DATA_BLOCK "DB2010_V"
TITLE = DB2010_V
{ S7_Optimized_Access := 'FALSE' }
AUTHOR : ABH
FAMILY : ZeusControl
VERSION : 1.0
//Bloique de datos valvula.
   STRUCT
      V { S7_SetPoint := 'False'} : Array[0.."N_MAX_DISP_V"] of "ZC_DISP_V";
      Mux { S7_SetPoint := 'False'} : Array[0.."N_MAX_MUX_DISP"] of "ZC_DISP_MUX_V";
      Agrup : Array[0.."N_MAX_DISP_AGRUP"] of "ZC_DISP_AGRUP";
   END_STRUCT;


BEGIN
   V[0].Hmi_Nombre := '';
   V[0].Hmi_Estado := 0;
   V[0].Estado_AutoMan := FALSE;
   V[0].Estado_Activado := FALSE;
   V[0].Estado_Enclavado := FALSE;
   V[0].Estado_EntradaRetornoReposo := FALSE;
   V[0].Estado_EntradaRetornoTrabajo := FALSE;
   V[0].Alarmas_Reposo := FALSE;
   V[0].Alarmas_Trabajo := FALSE;
   V[0].Alarmas_Mantenimiento := FALSE;
   V[0].Alarmas_Doble := FALSE;
   V[0].Alarmas_General := FALSE;
   V[0].Orden_ActivarManual := FALSE;
   V[0].Orden_ActivarAuto := TRUE;
   V[0].Orden_ResetCiclos := FALSE;
   V[0].Config_Habilitar := FALSE;
   V[0].Config_HabilitarRetornoReposo := TRUE;
   V[0].Config_HabilitarInvertirReposo := FALSE;
   V[0].Config_HabilitarRetornoTrabajo := TRUE;
   V[0].Config_HabilitarInvertirTrabajo := FALSE;
   V[0].Config_HabilitarMantenimiento := FALSE;
   V[0].Aux_oldActivado := FALSE;
   V[0].Aux_oldAlarma := FALSE;
   V[0].Aux_oldAutoMan := FALSE;
   V[0].Estado_SeguridadOk := TRUE;
   V[0].Config_GrupoAlarma := 0;
   V[0].Config_DireccionSalidaByte := 0;
   V[0].Config_DireccionSalidaBit := 0;
   V[0].Config_DireccionRetReposoByte := 0;
   V[0].Config_DireccionRetReposoBit := 0;
   V[0].Config_DireccionRetTrabajoByte := 0;
   V[0].Config_DireccionRetTrabajoBit := 0;
   V[0].Tiempos_SetPointTiempoAlarma := 10;
   V[0].Tiempos_Alarma := 0;
   V[0].Tiempos_SetPointCiclos := 1000;
   V[0].Tiempos_Ciclos := 0;
   V[1].Hmi_Nombre := 'VA-101';
   V[1].Hmi_Estado := 1;
   V[1].Estado_AutoMan := FALSE;
   V[1].Estado_Activado := FALSE;
   V[1].Estado_Enclavado := FALSE;
   V[1].Estado_EntradaRetornoReposo := FALSE;
   V[1].Estado_EntradaRetornoTrabajo := FALSE;
   V[1].Alarmas_Reposo := FALSE;
   V[1].Alarmas_Trabajo := FALSE;
   V[1].Alarmas_Mantenimiento := FALSE;
   V[1].Alarmas_Doble := FALSE;
   V[1].Alarmas_General := FALSE;
   V[1].Orden_ActivarManual := FALSE;
   V[1].Orden_ActivarAuto := FALSE;
   V[1].Orden_ResetCiclos := FALSE;
   V[1].Config_Habilitar := TRUE;
   V[1].Config_HabilitarRetornoReposo := FALSE;
   V[1].Config_HabilitarInvertirReposo := FALSE;
   V[1].Config_HabilitarRetornoTrabajo := TRUE;
   V[1].Config_HabilitarInvertirTrabajo := FALSE;
   V[1].Config_HabilitarMantenimiento := FALSE;
   V[1].Aux_oldActivado := FALSE;
   V[1].Aux_oldAlarma := FALSE;
   V[1].Aux_oldAutoMan := FALSE;
   V[1].Estado_SeguridadOk := TRUE;
   V[1].Config_GrupoAlarma := 0;
   V[1].Config_DireccionSalidaByte := 102;
   V[1].Config_DireccionSalidaBit := 0;
   V[1].Config_DireccionRetReposoByte := 0;
   V[1].Config_DireccionRetReposoBit := 0;
   V[1].Config_DireccionRetTrabajoByte := 102;
   V[1].Config_DireccionRetTrabajoBit := 0;
   V[1].Tiempos_SetPointTiempoAlarma := 10;
   V[1].Tiempos_Alarma := 0;
   V[1].Tiempos_SetPointCiclos := 1000;
   V[1].Tiempos_Ciclos := 66;
   V[2].Hmi_Nombre := 'VA-102';
   V[2].Hmi_Estado := 1;
   V[2].Estado_AutoMan := FALSE;
   V[2].Estado_Activado := FALSE;
   V[2].Estado_Enclavado := FALSE;
   V[2].Estado_EntradaRetornoReposo := FALSE;
   V[2].Estado_EntradaRetornoTrabajo := FALSE;
   V[2].Alarmas_Reposo := FALSE;
   V[2].Alarmas_Trabajo := FALSE;
   V[2].Alarmas_Mantenimiento := FALSE;
   V[2].Alarmas_Doble := FALSE;
   V[2].Alarmas_General := FALSE;
   V[2].Orden_ActivarManual := FALSE;
   V[2].Orden_ActivarAuto := FALSE;
   V[2].Orden_ResetCiclos := FALSE;
   V[2].Config_Habilitar := TRUE;
   V[2].Config_HabilitarRetornoReposo := FALSE;
   V[2].Config_HabilitarInvertirReposo := FALSE;
   V[2].Config_HabilitarRetornoTrabajo := TRUE;
   V[2].Config_HabilitarInvertirTrabajo := FALSE;
   V[2].Config_HabilitarMantenimiento := FALSE;
   V[2].Aux_oldActivado := FALSE;
   V[2].Aux_oldAlarma := FALSE;
   V[2].Aux_oldAutoMan := FALSE;
   V[2].Estado_SeguridadOk := TRUE;
   V[2].Config_GrupoAlarma := 0;
   V[2].Config_DireccionSalidaByte := 102;
   V[2].Config_DireccionSalidaBit := 1;
   V[2].Config_DireccionRetReposoByte := 0;
   V[2].Config_DireccionRetReposoBit := 0;
   V[2].Config_DireccionRetTrabajoByte := 102;
   V[2].Config_DireccionRetTrabajoBit := 1;
   V[2].Tiempos_SetPointTiempoAlarma := 10;
   V[2].Tiempos_Alarma := 0;
   V[2].Tiempos_SetPointCiclos := 1000;
   V[2].Tiempos_Ciclos := 104;
   V[3].Hmi_Nombre := 'VAD-103';
   V[3].Hmi_Estado := 1;
   V[3].Estado_AutoMan := FALSE;
   V[3].Estado_Activado := FALSE;
   V[3].Estado_Enclavado := FALSE;
   V[3].Estado_EntradaRetornoReposo := FALSE;
   V[3].Estado_EntradaRetornoTrabajo := FALSE;
   V[3].Alarmas_Reposo := FALSE;
   V[3].Alarmas_Trabajo := FALSE;
   V[3].Alarmas_Mantenimiento := FALSE;
   V[3].Alarmas_Doble := FALSE;
   V[3].Alarmas_General := FALSE;
   V[3].Orden_ActivarManual := FALSE;
   V[3].Orden_ActivarAuto := FALSE;
   V[3].Orden_ResetCiclos := FALSE;
   V[3].Config_Habilitar := TRUE;
   V[3].Config_HabilitarRetornoReposo := FALSE;
   V[3].Config_HabilitarInvertirReposo := FALSE;
   V[3].Config_HabilitarRetornoTrabajo := TRUE;
   V[3].Config_HabilitarInvertirTrabajo := FALSE;
   V[3].Config_HabilitarMantenimiento := FALSE;
   V[3].Aux_oldActivado := FALSE;
   V[3].Aux_oldAlarma := FALSE;
   V[3].Aux_oldAutoMan := FALSE;
   V[3].Estado_SeguridadOk := TRUE;
   V[3].Config_GrupoAlarma := 0;
   V[3].Config_DireccionSalidaByte := 102;
   V[3].Config_DireccionSalidaBit := 2;
   V[3].Config_DireccionRetReposoByte := 0;
   V[3].Config_DireccionRetReposoBit := 0;
   V[3].Config_DireccionRetTrabajoByte := 102;
   V[3].Config_DireccionRetTrabajoBit := 2;
   V[3].Tiempos_SetPointTiempoAlarma := 10;
   V[3].Tiempos_Alarma := 0;
   V[3].Tiempos_SetPointCiclos := 1000;
   V[3].Tiempos_Ciclos := 118;
   V[4].Hmi_Nombre := 'VAD-108';
   V[4].Hmi_Estado := 1;
   V[4].Estado_AutoMan := FALSE;
   V[4].Estado_Activado := FALSE;
   V[4].Estado_Enclavado := FALSE;
   V[4].Estado_EntradaRetornoReposo := FALSE;
   V[4].Estado_EntradaRetornoTrabajo := FALSE;
   V[4].Alarmas_Reposo := FALSE;
   V[4].Alarmas_Trabajo := FALSE;
   V[4].Alarmas_Mantenimiento := FALSE;
   V[4].Alarmas_Doble := FALSE;
   V[4].Alarmas_General := FALSE;
   V[4].Orden_ActivarManual := FALSE;
   V[4].Orden_ActivarAuto := FALSE;
   V[4].Orden_ResetCiclos := FALSE;
   V[4].Config_Habilitar := TRUE;
   V[4].Config_HabilitarRetornoReposo := FALSE;
   V[4].Config_HabilitarInvertirReposo := FALSE;
   V[4].Config_HabilitarRetornoTrabajo := TRUE;
   V[4].Config_HabilitarInvertirTrabajo := FALSE;
   V[4].Config_HabilitarMantenimiento := FALSE;
   V[4].Aux_oldActivado := FALSE;
   V[4].Aux_oldAlarma := FALSE;
   V[4].Aux_oldAutoMan := FALSE;
   V[4].Estado_SeguridadOk := TRUE;
   V[4].Config_GrupoAlarma := 0;
   V[4].Config_DireccionSalidaByte := 102;
   V[4].Config_DireccionSalidaBit := 3;
   V[4].Config_DireccionRetReposoByte := 0;
   V[4].Config_DireccionRetReposoBit := 0;
   V[4].Config_DireccionRetTrabajoByte := 102;
   V[4].Config_DireccionRetTrabajoBit := 3;
   V[4].Tiempos_SetPointTiempoAlarma := 10;
   V[4].Tiempos_Alarma := 0;
   V[4].Tiempos_SetPointCiclos := 1000;
   V[4].Tiempos_Ciclos := 28;
   V[5].Hmi_Nombre := 'VA-114';
   V[5].Hmi_Estado := 1;
   V[5].Estado_AutoMan := FALSE;
   V[5].Estado_Activado := FALSE;
   V[5].Estado_Enclavado := FALSE;
   V[5].Estado_EntradaRetornoReposo := FALSE;
   V[5].Estado_EntradaRetornoTrabajo := FALSE;
   V[5].Alarmas_Reposo := FALSE;
   V[5].Alarmas_Trabajo := FALSE;
   V[5].Alarmas_Mantenimiento := FALSE;
   V[5].Alarmas_Doble := FALSE;
   V[5].Alarmas_General := FALSE;
   V[5].Orden_ActivarManual := FALSE;
   V[5].Orden_ActivarAuto := FALSE;
   V[5].Orden_ResetCiclos := FALSE;
   V[5].Config_Habilitar := TRUE;
   V[5].Config_HabilitarRetornoReposo := FALSE;
   V[5].Config_HabilitarInvertirReposo := FALSE;
   V[5].Config_HabilitarRetornoTrabajo := TRUE;
   V[5].Config_HabilitarInvertirTrabajo := FALSE;
   V[5].Config_HabilitarMantenimiento := FALSE;
   V[5].Aux_oldActivado := FALSE;
   V[5].Aux_oldAlarma := FALSE;
   V[5].Aux_oldAutoMan := FALSE;
   V[5].Estado_SeguridadOk := TRUE;
   V[5].Config_GrupoAlarma := 0;
   V[5].Config_DireccionSalidaByte := 102;
   V[5].Config_DireccionSalidaBit := 4;
   V[5].Config_DireccionRetReposoByte := 0;
   V[5].Config_DireccionRetReposoBit := 0;
   V[5].Config_DireccionRetTrabajoByte := 102;
   V[5].Config_DireccionRetTrabajoBit := 4;
   V[5].Tiempos_SetPointTiempoAlarma := 10;
   V[5].Tiempos_Alarma := 0;
   V[5].Tiempos_SetPointCiclos := 1000;
   V[5].Tiempos_Ciclos := 6;
   V[6].Hmi_Nombre := 'VA3-115';
   V[6].Hmi_Estado := 1;
   V[6].Estado_AutoMan := FALSE;
   V[6].Estado_Activado := FALSE;
   V[6].Estado_Enclavado := FALSE;
   V[6].Estado_EntradaRetornoReposo := FALSE;
   V[6].Estado_EntradaRetornoTrabajo := FALSE;
   V[6].Alarmas_Reposo := FALSE;
   V[6].Alarmas_Trabajo := FALSE;
   V[6].Alarmas_Mantenimiento := FALSE;
   V[6].Alarmas_Doble := FALSE;
   V[6].Alarmas_General := FALSE;
   V[6].Orden_ActivarManual := FALSE;
   V[6].Orden_ActivarAuto := FALSE;
   V[6].Orden_ResetCiclos := FALSE;
   V[6].Config_Habilitar := TRUE;
   V[6].Config_HabilitarRetornoReposo := FALSE;
   V[6].Config_HabilitarInvertirReposo := FALSE;
   V[6].Config_HabilitarRetornoTrabajo := TRUE;
   V[6].Config_HabilitarInvertirTrabajo := FALSE;
   V[6].Config_HabilitarMantenimiento := FALSE;
   V[6].Aux_oldActivado := FALSE;
   V[6].Aux_oldAlarma := FALSE;
   V[6].Aux_oldAutoMan := FALSE;
   V[6].Estado_SeguridadOk := TRUE;
   V[6].Config_GrupoAlarma := 0;
   V[6].Config_DireccionSalidaByte := 102;
   V[6].Config_DireccionSalidaBit := 5;
   V[6].Config_DireccionRetReposoByte := 0;
   V[6].Config_DireccionRetReposoBit := 0;
   V[6].Config_DireccionRetTrabajoByte := 102;
   V[6].Config_DireccionRetTrabajoBit := 5;
   V[6].Tiempos_SetPointTiempoAlarma := 10;
   V[6].Tiempos_Alarma := 0;
   V[6].Tiempos_SetPointCiclos := 1000;
   V[6].Tiempos_Ciclos := 6;
   V[7].Hmi_Nombre := 'VA3-116';
   V[7].Hmi_Estado := 1;
   V[7].Estado_AutoMan := FALSE;
   V[7].Estado_Activado := FALSE;
   V[7].Estado_Enclavado := FALSE;
   V[7].Estado_EntradaRetornoReposo := FALSE;
   V[7].Estado_EntradaRetornoTrabajo := FALSE;
   V[7].Alarmas_Reposo := FALSE;
   V[7].Alarmas_Trabajo := FALSE;
   V[7].Alarmas_Mantenimiento := FALSE;
   V[7].Alarmas_Doble := FALSE;
   V[7].Alarmas_General := FALSE;
   V[7].Orden_ActivarManual := FALSE;
   V[7].Orden_ActivarAuto := FALSE;
   V[7].Orden_ResetCiclos := FALSE;
   V[7].Config_Habilitar := TRUE;
   V[7].Config_HabilitarRetornoReposo := FALSE;
   V[7].Config_HabilitarInvertirReposo := FALSE;
   V[7].Config_HabilitarRetornoTrabajo := TRUE;
   V[7].Config_HabilitarInvertirTrabajo := FALSE;
   V[7].Config_HabilitarMantenimiento := FALSE;
   V[7].Aux_oldActivado := FALSE;
   V[7].Aux_oldAlarma := FALSE;
   V[7].Aux_oldAutoMan := FALSE;
   V[7].Estado_SeguridadOk := TRUE;
   V[7].Config_GrupoAlarma := 0;
   V[7].Config_DireccionSalidaByte := 102;
   V[7].Config_DireccionSalidaBit := 6;
   V[7].Config_DireccionRetReposoByte := 0;
   V[7].Config_DireccionRetReposoBit := 0;
   V[7].Config_DireccionRetTrabajoByte := 102;
   V[7].Config_DireccionRetTrabajoBit := 6;
   V[7].Tiempos_SetPointTiempoAlarma := 10;
   V[7].Tiempos_Alarma := 0;
   V[7].Tiempos_SetPointCiclos := 1000;
   V[7].Tiempos_Ciclos := 6;
   V[8].Hmi_Nombre := 'VAD-117';
   V[8].Hmi_Estado := 1;
   V[8].Estado_AutoMan := FALSE;
   V[8].Estado_Activado := FALSE;
   V[8].Estado_Enclavado := FALSE;
   V[8].Estado_EntradaRetornoReposo := FALSE;
   V[8].Estado_EntradaRetornoTrabajo := FALSE;
   V[8].Alarmas_Reposo := FALSE;
   V[8].Alarmas_Trabajo := FALSE;
   V[8].Alarmas_Mantenimiento := FALSE;
   V[8].Alarmas_Doble := FALSE;
   V[8].Alarmas_General := FALSE;
   V[8].Orden_ActivarManual := FALSE;
   V[8].Orden_ActivarAuto := FALSE;
   V[8].Orden_ResetCiclos := FALSE;
   V[8].Config_Habilitar := TRUE;
   V[8].Config_HabilitarRetornoReposo := FALSE;
   V[8].Config_HabilitarInvertirReposo := FALSE;
   V[8].Config_HabilitarRetornoTrabajo := TRUE;
   V[8].Config_HabilitarInvertirTrabajo := FALSE;
   V[8].Config_HabilitarMantenimiento := FALSE;
   V[8].Aux_oldActivado := FALSE;
   V[8].Aux_oldAlarma := FALSE;
   V[8].Aux_oldAutoMan := FALSE;
   V[8].Estado_SeguridadOk := TRUE;
   V[8].Config_GrupoAlarma := 0;
   V[8].Config_DireccionSalidaByte := 102;
   V[8].Config_DireccionSalidaBit := 7;
   V[8].Config_DireccionRetReposoByte := 0;
   V[8].Config_DireccionRetReposoBit := 0;
   V[8].Config_DireccionRetTrabajoByte := 102;
   V[8].Config_DireccionRetTrabajoBit := 7;
   V[8].Tiempos_SetPointTiempoAlarma := 10;
   V[8].Tiempos_Alarma := 0;
   V[8].Tiempos_SetPointCiclos := 1000;
   V[8].Tiempos_Ciclos := 84;
   V[9].Hmi_Nombre := 'VAD-120';
   V[9].Hmi_Estado := 1;
   V[9].Estado_AutoMan := FALSE;
   V[9].Estado_Activado := FALSE;
   V[9].Estado_Enclavado := FALSE;
   V[9].Estado_EntradaRetornoReposo := FALSE;
   V[9].Estado_EntradaRetornoTrabajo := FALSE;
   V[9].Alarmas_Reposo := FALSE;
   V[9].Alarmas_Trabajo := FALSE;
   V[9].Alarmas_Mantenimiento := FALSE;
   V[9].Alarmas_Doble := FALSE;
   V[9].Alarmas_General := FALSE;
   V[9].Orden_ActivarManual := FALSE;
   V[9].Orden_ActivarAuto := FALSE;
   V[9].Orden_ResetCiclos := FALSE;
   V[9].Config_Habilitar := TRUE;
   V[9].Config_HabilitarRetornoReposo := FALSE;
   V[9].Config_HabilitarInvertirReposo := FALSE;
   V[9].Config_HabilitarRetornoTrabajo := TRUE;
   V[9].Config_HabilitarInvertirTrabajo := FALSE;
   V[9].Config_HabilitarMantenimiento := FALSE;
   V[9].Aux_oldActivado := FALSE;
   V[9].Aux_oldAlarma := FALSE;
   V[9].Aux_oldAutoMan := FALSE;
   V[9].Estado_SeguridadOk := TRUE;
   V[9].Config_GrupoAlarma := 0;
   V[9].Config_DireccionSalidaByte := 103;
   V[9].Config_DireccionSalidaBit := 0;
   V[9].Config_DireccionRetReposoByte := 0;
   V[9].Config_DireccionRetReposoBit := 0;
   V[9].Config_DireccionRetTrabajoByte := 103;
   V[9].Config_DireccionRetTrabajoBit := 0;
   V[9].Tiempos_SetPointTiempoAlarma := 10;
   V[9].Tiempos_Alarma := 0;
   V[9].Tiempos_SetPointCiclos := 1000;
   V[9].Tiempos_Ciclos := 28;
   V[10].Hmi_Nombre := 'VA-126';
   V[10].Hmi_Estado := 1;
   V[10].Estado_AutoMan := FALSE;
   V[10].Estado_Activado := FALSE;
   V[10].Estado_Enclavado := FALSE;
   V[10].Estado_EntradaRetornoReposo := FALSE;
   V[10].Estado_EntradaRetornoTrabajo := FALSE;
   V[10].Alarmas_Reposo := FALSE;
   V[10].Alarmas_Trabajo := FALSE;
   V[10].Alarmas_Mantenimiento := FALSE;
   V[10].Alarmas_Doble := FALSE;
   V[10].Alarmas_General := FALSE;
   V[10].Orden_ActivarManual := FALSE;
   V[10].Orden_ActivarAuto := FALSE;
   V[10].Orden_ResetCiclos := FALSE;
   V[10].Config_Habilitar := TRUE;
   V[10].Config_HabilitarRetornoReposo := FALSE;
   V[10].Config_HabilitarInvertirReposo := FALSE;
   V[10].Config_HabilitarRetornoTrabajo := TRUE;
   V[10].Config_HabilitarInvertirTrabajo := FALSE;
   V[10].Config_HabilitarMantenimiento := FALSE;
   V[10].Aux_oldActivado := FALSE;
   V[10].Aux_oldAlarma := FALSE;
   V[10].Aux_oldAutoMan := FALSE;
   V[10].Estado_SeguridadOk := TRUE;
   V[10].Config_GrupoAlarma := 0;
   V[10].Config_DireccionSalidaByte := 103;
   V[10].Config_DireccionSalidaBit := 1;
   V[10].Config_DireccionRetReposoByte := 0;
   V[10].Config_DireccionRetReposoBit := 0;
   V[10].Config_DireccionRetTrabajoByte := 103;
   V[10].Config_DireccionRetTrabajoBit := 1;
   V[10].Tiempos_SetPointTiempoAlarma := 10;
   V[10].Tiempos_Alarma := 0;
   V[10].Tiempos_SetPointCiclos := 1000;
   V[10].Tiempos_Ciclos := 70;
   Mux[0].Habilitar := TRUE;
   Mux[0].ExisteCambio := FALSE;
   Mux[0].MaxVisible := FALSE;
   Mux[0].Index := 182;
   Mux[0].oldIndex := 182;
   Mux[0].V.Hmi_Nombre := 'VA-438';
   Mux[0].V.Hmi_Estado := 1;
   Mux[0].V.Estado_AutoMan := FALSE;
   Mux[0].V.Estado_Activado := FALSE;
   Mux[0].V.Estado_Enclavado := FALSE;
   Mux[0].V.Estado_EntradaRetornoReposo := FALSE;
   Mux[0].V.Estado_EntradaRetornoTrabajo := FALSE;
   Mux[0].V.Alarmas_Reposo := FALSE;
   Mux[0].V.Alarmas_Trabajo := FALSE;
   Mux[0].V.Alarmas_Mantenimiento := FALSE;
   Mux[0].V.Alarmas_Doble := FALSE;
   Mux[0].V.Alarmas_General := FALSE;
   Mux[0].V.Orden_ActivarManual := FALSE;
   Mux[0].V.Orden_ActivarAuto := FALSE;
   Mux[0].V.Orden_ResetCiclos := FALSE;
   Mux[0].V.Config_Habilitar := TRUE;
   Mux[0].V.Config_HabilitarRetornoReposo := FALSE;
   Mux[0].V.Config_HabilitarInvertirReposo := FALSE;
   Mux[0].V.Config_HabilitarRetornoTrabajo := FALSE;
   Mux[0].V.Config_HabilitarInvertirTrabajo := FALSE;
   Mux[0].V.Config_HabilitarMantenimiento := FALSE;
   Mux[0].V.Aux_oldActivado := FALSE;
   Mux[0].V.Aux_oldAlarma := FALSE;
   Mux[0].V.Aux_oldAutoMan := FALSE;
   Mux[0].V.Estado_SeguridadOk := TRUE;
   Mux[0].V.Config_GrupoAlarma := 2;
   Mux[0].V.Config_DireccionSalidaByte := 325;
   Mux[0].V.Config_DireccionSalidaBit := 2;
   Mux[0].V.Config_DireccionRetReposoByte := 0;
   Mux[0].V.Config_DireccionRetReposoBit := 0;
   Mux[0].V.Config_DireccionRetTrabajoByte := 0;
   Mux[0].V.Config_DireccionRetTrabajoBit := 0;
   Mux[0].V.Tiempos_SetPointTiempoAlarma := 10;
   Mux[0].V.Tiempos_Alarma := 0;
   Mux[0].V.Tiempos_SetPointCiclos := 1000;
   Mux[0].V.Tiempos_Ciclos := 1200;
   Mux[1].Habilitar := TRUE;
   Mux[1].ExisteCambio := FALSE;
   Mux[1].MaxVisible := FALSE;
   Mux[1].Index := 0;
   Mux[1].oldIndex := 0;
   Mux[1].V.Hmi_Nombre := '';
   Mux[1].V.Hmi_Estado := 0;
   Mux[1].V.Estado_AutoMan := FALSE;
   Mux[1].V.Estado_Activado := FALSE;
   Mux[1].V.Estado_Enclavado := FALSE;
   Mux[1].V.Estado_EntradaRetornoReposo := FALSE;
   Mux[1].V.Estado_EntradaRetornoTrabajo := FALSE;
   Mux[1].V.Alarmas_Reposo := FALSE;
   Mux[1].V.Alarmas_Trabajo := FALSE;
   Mux[1].V.Alarmas_Mantenimiento := FALSE;
   Mux[1].V.Alarmas_Doble := FALSE;
   Mux[1].V.Alarmas_General := FALSE;
   Mux[1].V.Orden_ActivarManual := FALSE;
   Mux[1].V.Orden_ActivarAuto := TRUE;
   Mux[1].V.Orden_ResetCiclos := FALSE;
   Mux[1].V.Config_Habilitar := FALSE;
   Mux[1].V.Config_HabilitarRetornoReposo := TRUE;
   Mux[1].V.Config_HabilitarInvertirReposo := FALSE;
   Mux[1].V.Config_HabilitarRetornoTrabajo := TRUE;
   Mux[1].V.Config_HabilitarInvertirTrabajo := FALSE;
   Mux[1].V.Config_HabilitarMantenimiento := FALSE;
   Mux[1].V.Aux_oldActivado := FALSE;
   Mux[1].V.Aux_oldAlarma := FALSE;
   Mux[1].V.Aux_oldAutoMan := FALSE;
   Mux[1].V.Estado_SeguridadOk := TRUE;
   Mux[1].V.Config_GrupoAlarma := 0;
   Mux[1].V.Config_DireccionSalidaByte := 0;
   Mux[1].V.Config_DireccionSalidaBit := 0;
   Mux[1].V.Config_DireccionRetReposoByte := 0;
   Mux[1].V.Config_DireccionRetReposoBit := 0;
   Mux[1].V.Config_DireccionRetTrabajoByte := 0;
   Mux[1].V.Config_DireccionRetTrabajoBit := 0;
   Mux[1].V.Tiempos_SetPointTiempoAlarma := 10;
   Mux[1].V.Tiempos_Alarma := 0;
   Mux[1].V.Tiempos_SetPointCiclos := 1000;
   Mux[1].V.Tiempos_Ciclos := 0;
   Mux[2].Habilitar := TRUE;
   Mux[2].ExisteCambio := FALSE;
   Mux[2].MaxVisible := FALSE;
   Mux[2].Index := 0;
   Mux[2].oldIndex := 0;
   Mux[2].V.Hmi_Nombre := '';
   Mux[2].V.Hmi_Estado := 0;
   Mux[2].V.Estado_AutoMan := FALSE;
   Mux[2].V.Estado_Activado := FALSE;
   Mux[2].V.Estado_Enclavado := FALSE;
   Mux[2].V.Estado_EntradaRetornoReposo := FALSE;
   Mux[2].V.Estado_EntradaRetornoTrabajo := FALSE;
   Mux[2].V.Alarmas_Reposo := FALSE;
   Mux[2].V.Alarmas_Trabajo := FALSE;
   Mux[2].V.Alarmas_Mantenimiento := FALSE;
   Mux[2].V.Alarmas_Doble := FALSE;
   Mux[2].V.Alarmas_General := FALSE;
   Mux[2].V.Orden_ActivarManual := FALSE;
   Mux[2].V.Orden_ActivarAuto := TRUE;
   Mux[2].V.Orden_ResetCiclos := FALSE;
   Mux[2].V.Config_Habilitar := FALSE;
   Mux[2].V.Config_HabilitarRetornoReposo := TRUE;
   Mux[2].V.Config_HabilitarInvertirReposo := FALSE;
   Mux[2].V.Config_HabilitarRetornoTrabajo := TRUE;
   Mux[2].V.Config_HabilitarInvertirTrabajo := FALSE;
   Mux[2].V.Config_HabilitarMantenimiento := FALSE;
   Mux[2].V.Aux_oldActivado := FALSE;
   Mux[2].V.Aux_oldAlarma := FALSE;
   Mux[2].V.Aux_oldAutoMan := FALSE;
   Mux[2].V.Estado_SeguridadOk := TRUE;
   Mux[2].V.Config_GrupoAlarma := 0;
   Mux[2].V.Config_DireccionSalidaByte := 0;
   Mux[2].V.Config_DireccionSalidaBit := 0;
   Mux[2].V.Config_DireccionRetReposoByte := 0;
   Mux[2].V.Config_DireccionRetReposoBit := 0;
   Mux[2].V.Config_DireccionRetTrabajoByte := 0;
   Mux[2].V.Config_DireccionRetTrabajoBit := 0;
   Mux[2].V.Tiempos_SetPointTiempoAlarma := 10;
   Mux[2].V.Tiempos_Alarma := 0;
   Mux[2].V.Tiempos_SetPointCiclos := 1000;
   Mux[2].V.Tiempos_Ciclos := 0;
   Agrup[0].AlgunaEnManual := FALSE;
   Agrup[0].AlgunaAlarma := FALSE;
   Agrup[0].NuevaAlarma := FALSE;
   Agrup[1].AlgunaEnManual := TRUE;
   Agrup[1].AlgunaAlarma := FALSE;
   Agrup[1].NuevaAlarma := FALSE;

END_DATA_BLOCK

